PROGRAM MAIN_FS
VAR
	i_xFFReset: INT;
END_VAR

(*
PA1L0_VFS_01(
	i_xPMPS_OK:= TRUE, 
	i_xExt_OK:= TRUE, 
	io_fbFFHWO:= g_FastFaultOutput3);
*)	
TV3L0_VFS_01(
	i_xPMPS_OK:= TRUE, 
	i_xExt_OK:= TRUE, 
	io_fbFFHWO:= g_FastFaultOutput3);

(*FastFaultOuput*)	
g_FastFaultOutput3.Execute(bAutoReset:= TRUE);

END_PROGRAM

(* stored: Version 1.1.0.1, ProductVersion 3.1.4022.18
   POU MAIN_FS: Id {cd87fa27-2963-491a-8560-055b56a6fb32}, SpecialFunc None *)
